// Mitsubishi GX Works2 project: 1축 기구 jog 운전 제어   PLC: Q02/Q02H

PROGRAM MAIN
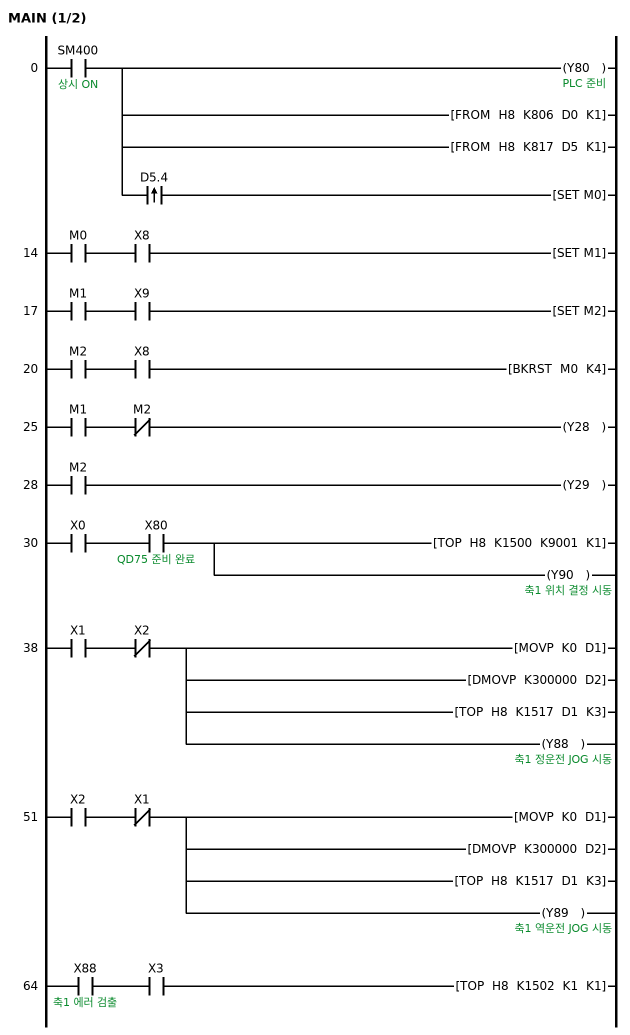
0     LD      SM400  ; 상시 ON
      OUT     Y80  ; PLC 준비
      FROM    H8 K806 D0 K1
      FROM    H8 K817 D5 K1
      ANDP    D5.4
      SET     M0
14    LD      M0
      AND     X8
      SET     M1
17    LD      M1
      AND     X9
      SET     M2
20    LD      M2
      AND     X8
      BKRST   M0 K4
25    LD      M1
      ANI     M2
      OUT     Y28
28    LD      M2
      OUT     Y29
30    LD      X0
      AND     X80  ; QD75 준비 완료
      TOP     H8 K1500 K9001 K1
      OUT     Y90  ; 축1 위치 결정 시동
38    LD      X1
      ANI     X2
      MOVP    K0 D1
      DMOVP   K300000 D2
      TOP     H8 K1517 D1 K3
      OUT     Y88  ; 축1 정운전 JOG 시동
51    LD      X2
      ANI     X1
      MOVP    K0 D1
      DMOVP   K300000 D2
      TOP     H8 K1517 D1 K3
      OUT     Y89  ; 축1 역운전 JOG 시동
64    LD      X88  ; 축1 에러 검출
      AND     X3
      TOP     H8 K1502 K1 K1
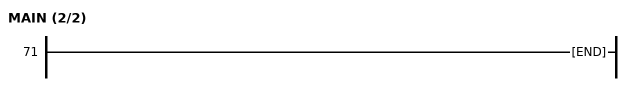
71    END
END_PROGRAM

// device comments not shown above
X81  ; 동기용 플래그
X84  ; 축1 M 코드 ON
X8C  ; 축1 BUSY
X90  ; 축1 시동 완료
X94  ; 축1 위치 결정 완료
Y84  ; 축1 축 정지
Y94  ; 축1 실행 금지 플래그
